SUBAPPLICATION GreenWhiteBackground_Verteiler_heben (* Subapplication Type *)
  (* Standard: 61499-2 *)
  (* Version 1.0, 2023-02-11, franz *)
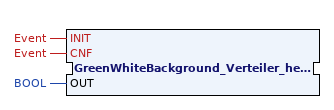
  EVENT_INPUT
    INIT;
    CNF;
  END_EVENT
  VAR_INPUT
    OUT : BOOL;
  END_VAR
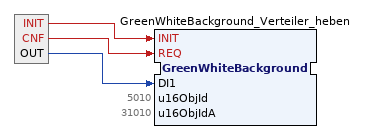
  SUBAPPS
    GreenWhiteBackground_Verteiler_heben : GreenWhiteBackground(u16ObjId := 5010, u16ObjIdA := 31010);
  END_SUBAPPS
  EVENT_CONNECTIONS
    INIT TO GreenWhiteBackground_Verteiler_heben.INIT;
    CNF TO GreenWhiteBackground_Verteiler_heben.REQ;
  END_CONNECTIONS
  DATA_CONNECTIONS
    OUT TO GreenWhiteBackground_Verteiler_heben.DI1;
  END_CONNECTIONS
END_SUBAPPLICATION
